// TIA Portal V19 export
DATA_BLOCK "A0302_Mng_BtrkListToCheck"   // DB182
// stored: InstanceOfName A0302_Mng_BtrkListToCheck_FB, InstanceOfType FB
"A0302_Mng_BtrkListToCheck_FB"
   // VAR_IN_OUT
   //    BTrk : Array[1.."BTRK_A03_EXIT_TOCHECK_ITEMS"] of "BTrk_item";
   //    FullList : Bool;
   // END_VAR
   // VAR
   //    i { ExternalAccessible := 'False'; ExternalVisible := 'False'; ExternalWritable := 'False'} : Int;
   //    j : Int;
   //    Control : Struct
   //       NoPlaceEmpty : USInt;
   //       StopCount : Bool;
   //       Pls_ClearArchive : Bool;
   //    END_STRUCT;
   // END_VAR
BEGIN
END_DATA_BLOCK
